// TIA Portal V20 export
DATA_BLOCK "BK25"   // DB272
// stored: MemoryReserve 100
   VAR
      "X10-1 TOP TAPE ATTACHMENT #1 VACUUM ON" : Bool;
      "X10-2 TOP TAPE ATTACHMENT #1 VACUUM OFF" : Bool;
      "X12-1 SPARE" : Bool;
      "X12-2 SPARE" : Bool;
      "X14-1 SPARE" : Bool;
      "X14-2 SPARE" : Bool;
      "X16-1 SPARE" : Bool;
      "X16-2 SPARE" : Bool;
   END_VAR
BEGIN
END_DATA_BLOCK
